// TIA Portal project "scl_10" (V18)

(* hardware
DEVICE "S7-1200 station_1"  S7-1200 Station
   slot 0: "Rack_0"  S7-1200 Rack  Rack  V1.0
   slot 1: "PLC_1"  CPU 1214C DC/DC/DC  6ES7 214-1AG40-0XB0  V4.6
*)

// ===== PLC "PLC_1"  CPU 1214C DC/DC/DC =====

VAR_GLOBAL   // PLC tag table "Default tag table"
   "START" AT %I0.0 : Bool;
   "STOP" AT %I0.1 : Bool;
   "SAYMA ALANI" AT %MW30 : UInt;
   "DONGU SAYISI" AT %MW32 : UInt;
   "DARBE MERKER" AT %Q0.3 : Bool;
   "YARDIMCI DARBE MERKE" AT %M0.0 : Bool;
   "ÇIKIŞ" AT %Q0.0 : Bool;
END_VAR

FUNCTION "Block_1" : Void   // FC1, SCL
{ S7_Optimized_Access := 'TRUE' }
VERSION : 0.1
BEGIN
   "DARBE MERKER" := "START" AND NOT "YARDIMCI DARBE MERKE";
   "YARDIMCI DARBE MERKE" := "START";
   IF "DARBE MERKER" THEN

       REPEAT
           "SAYMA ALANI" := "SAYMA ALANI" + 10;

       UNTIL "SAYMA ALANI">=400 END_REPEAT;



   END_IF;

   IF "SAYMA ALANI" > 1200 THEN
       "ÇIKIŞ" := 1;

   END_IF;

   IF "ÇIKIŞ" = 1 THEN
       "ÇIKIŞ" := 0;
       "SAYMA ALANI" := 0;
   END_IF;
END_FUNCTION

ORGANIZATION_BLOCK "Main"   // OB1, LAD, ProgramCycle
TITLE = "Main Program Sweep (Cycle)"
{ S7_Optimized_Access := 'TRUE' }
VERSION : 0.1
   VAR_INPUT
      Initial_Call : Bool;   // Initial call of this OB
      Remanence : Bool;   // =True, if remanent data are available
   END_VAR
BEGIN
END_ORGANIZATION_BLOCK